FUNCTION convertToHodnota : REAL

VAR_INPUT
	pCommand	:	REAL;
	enaPosDir	:	BOOL;
END_VAR

//	mA  conversion  in  0 to 1000
IF  enaPosDir THEN
	convertToHodnota := (pCommand * (generalVariable.conParammetr.CurPosDirMax - generalVariable.conParammetr.CurPosDirMin)/1000) + generalVariable.conParammetr.CurPosDirMin;
	ELSE
		convertToHodnota := (pCommand * (generalVariable.conParammetr.CurNegDirMax - generalVariable.conParammetr.CurNegDirMin)/1000) + generalVariable.conParammetr.CurNegDirMin;
		END_IF;

END_FUNCTION

(* stored: Version 1.1.0.1, ProductVersion 3.1.4024.12
   POU convertToHodnota: Id {0b0224bc-4975-4099-9840-bb6086fabaa8}, SpecialFunc None *)
